(* PLC project Unnamed, Unknown Unnamed 1 *)
(* stored: creationDateTime 2023-03-10T10:37:17, modificationDateTime 2023-03-15T15:56:42 *)

(* ISBN: 978-3-8085-3450-2, Aufgabe 9 *)
FUNCTION_BLOCK Santa_Claus_Doll_Rope_Winch
  VAR_INPUT
    INS1 : BOOL;
    INB1 : BOOL;
    INB2 : BOOL;
  END_VAR
  VAR_OUTPUT
    OUT1 : BOOL;
    OUT2 : BOOL;
  END_VAR
  VAR
    ME1 : BOOL;
    ME2 : BOOL;
  END_VAR
  VAR  (* added by the conversion: wires and edge detectors of the diagram *)
    _NOT11_OUT : BOOL;
    _NOT9_OUT : BOOL;
    _AND13_OUT : BOOL;
    _AND19_OUT : BOOL;
  END_VAR

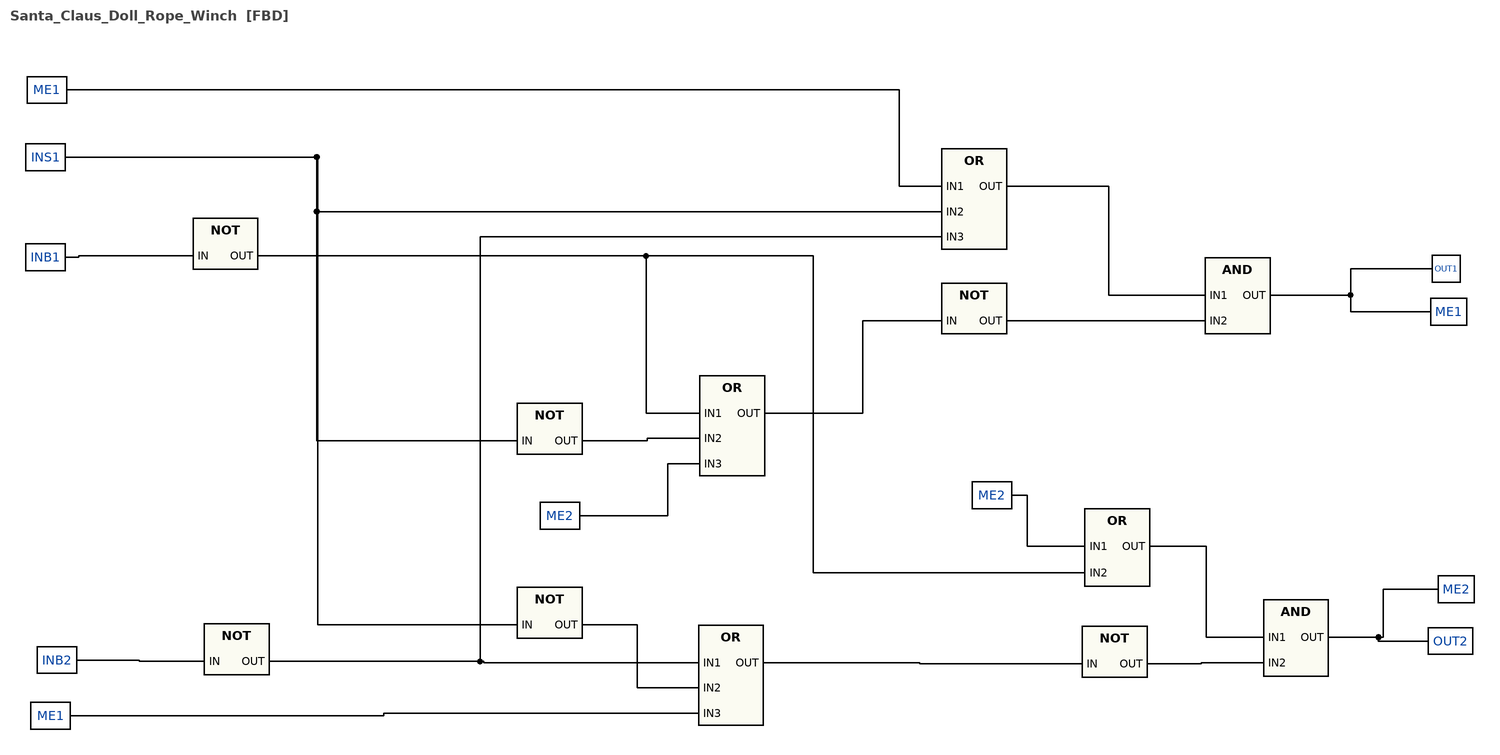
(* FBD diagram, written out as Structured Text *)
_NOT11_OUT := NOT INB2;
_NOT9_OUT := NOT INB1;
_AND13_OUT := (ME1 OR INS1 OR _NOT11_OUT) AND NOT (_NOT9_OUT OR NOT INS1 OR ME2);
OUT1 := _AND13_OUT;
ME1 := _AND13_OUT;
_AND19_OUT := (ME2 OR _NOT9_OUT) AND NOT (_NOT11_OUT OR NOT INS1 OR ME1);
ME2 := _AND19_OUT;
OUT2 := _AND19_OUT;
END_FUNCTION_BLOCK

CONFIGURATION config
  RESOURCE resource1 ON PLC
  END_RESOURCE
END_CONFIGURATION
